(*			
	RAFALOS
	Rafał Osajda		19.09.2025		TC 4024.66
	Rodzic dla wszystkich podzespołów głównych w maszynie 
*)
FUNCTION_BLOCK FB_BaseTopElement EXTENDS FB_BaseGroupElement IMPLEMENTS ITF_BaseTopElement, ITF_BaseTopElement_HMI_Connector
VAR
END_VAR

METHOD FB_init : BOOL
VAR_INPUT
	bInitRetains : BOOL; // if TRUE, the retain variables are initialized (warm start / cold start)
	bInCopyCode : BOOL;  // if TRUE, the instance afterwards gets moved into the copy code (online change)
END_VAR
THIS^.stIdentifier.eType			:= E_BaseElementType.eTop;
END_METHOD

METHOD PUBLIC PierwszePrzejscie : BOOL
VAR_INPUT
END_VAR
END_METHOD

END_FUNCTION_BLOCK

(* stored: Version 1.1.0.1
   POU FB_BaseTopElement: Id {b23ea2e3-7979-0bc9-362e-7cf0941731d6}, SpecialFunc None
   Method FB_init: Id {8200787b-ee94-0c86-2812-2a65b9019324}
   Method PierwszePrzejscie: Id {6e135063-cf1d-0182-35da-13dbdee6cbc3} *)
